FUNCTION_BLOCK RFID_Test EXTENDS TcUnit.FB_TestSuite

END_FUNCTION_BLOCK

(* stored: Version 1.1.0.1, ProductVersion 3.1.4024.12
   POU RFID_Test: Id {4bc4c850-1311-0ca8-1d83-9cb8e9140fb1}, SpecialFunc None *)
